(* PLC project tapis, TNI-Software ControlBuild 4.00 *)
(* stored: creationDateTime 2018-09-17T17:24:47-01:00 *)

FUNCTION_BLOCK tapis_conv.tapis
  VAR_INPUT  (* CB.kind=inputVars *)
    Marche : BOOL := false;
  END_VAR
  VAR_OUTPUT  (* CB.kind=outputVars *)
    Deplacement : REAL := 0.0;
  END_VAR

if Marche=true 
then 
	while Deplacement<50 DO
		Deplacement:=Deplacement+0.1;
		EXIT;
	end_while;
end_if;
END_FUNCTION_BLOCK
